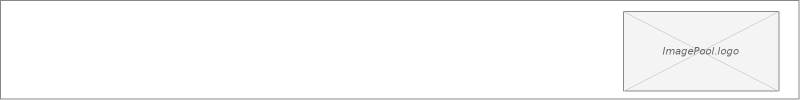
VISUALIZATION Header  // 800x100
    Image (623,11 156x80), image: ImagePool.logo
END_VISUALIZATION

(* stored: Version 1.1.0.1, ProductVersion 3.1.4024.12
   Visu Header: Id {3dd4e1e5-74e9-4840-87eb-4dfeda43e721} *)
